TYPE AX52XXDriveStatuses :
STRUCT
	///Is the drive in a busy state?
	busyStatus: BusyStatus;
	///Is the drive in a healthy state?
	healthStatus: HealthStatus;
END_STRUCT
END_TYPE

(* stored: Version 1.1.0.1, ProductVersion 3.1.4019.2
   DUT AX52XXDriveStatuses: Id {b01749c9-03d2-4fe7-8f10-afd18b6081d4} *)
